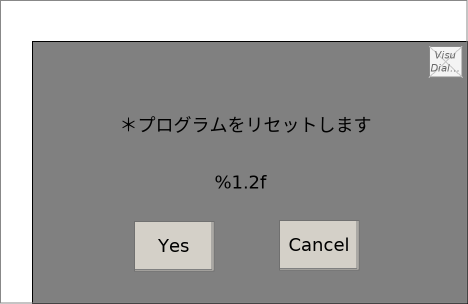
VISUALIZATION d_resetProject  // 468x304
    Rectangle (32,41 436x263)
    Image (429,46 33x31), image: VisuDialogs.ImagePoolDialogs.Delete
        OnMouseClick: CloseDialog Dialog=d_resetProject, Result=OK, NumpadKeypadSet=True
        OnMouseClick: execute { gvl_visu.flg_btn_projectReset := FALSE; }
    Label (57,93 377x65), "＊プログラムをリセットします"
    Button (134,221 80x50), "Yes", colour toggle: gvl_visu.flg_btn_projectReset
        toggle gvl_visu.flg_btn_projectReset
    Button (279,220 80x50), "Cancel"
        OnMouseClick: CloseDialog Dialog=d_resetProject, Result=OK, NumpadKeypadSet=True
        OnMouseClick: execute { gvl_visu.flg_btn_projectReset := FALSE; }
    Rectangle (53,157 370x51), "%1.2f", text variable: gvl_visu.var_projectResetLastTime
END_VISUALIZATION

(* stored: Version 1.1.0.1, ProductVersion 3.1.4024.12
   Visu d_resetProject: Id {7287312f-7bee-44bb-8230-09b6744873fe} *)
